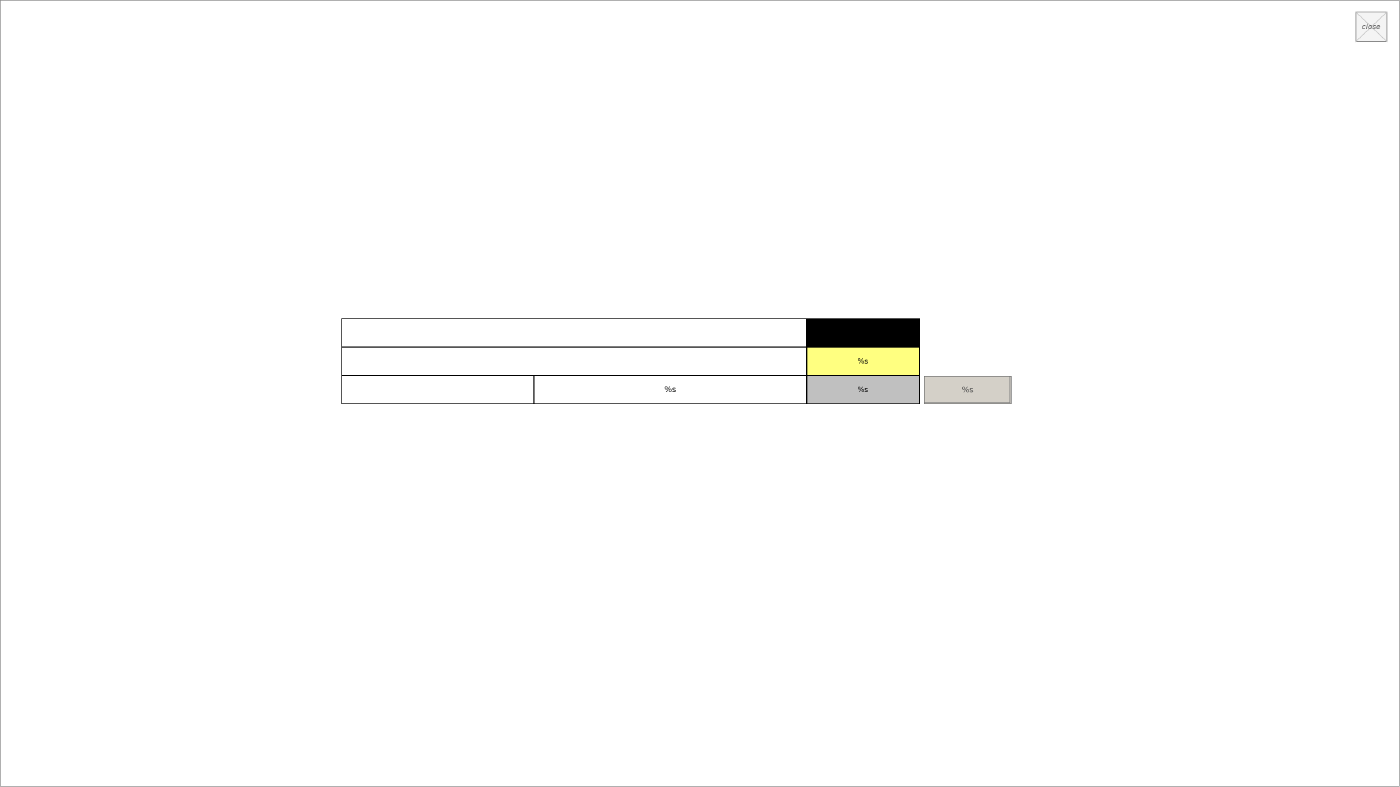
VISUALIZATION VISU_CONFIG_ECOMODE  // 1920x1080, background image fond_blanc_1280_1024
    Rectangle (468,476 638x39), text list: 'TextList_EcoMode', text index: 1
    Rectangle (468,437 638x39), text list: 'TextList_EcoMode', text index: 0
    Rectangle (468,515 264x39), text list: 'TextList_EcoMode', text index: 2
    Rectangle (1106,476 155x39), "%s", text variable: .MACHINE.CONF_Tps_Inactivite, input disabled if: NOT Global_Variables.PRG_USER.ACTU_USER.CONF_MACHINE
        OnMouseClick: write the text variable via InputWithLimits, min 0
    Rectangle (1106,437 155x39), colour toggle: MACHINE.CONF_Standby_Auto, input disabled if: NOT Global_Variables.PRG_USER.ACTU_USER.CONF_MACHINE
        toggle MACHINE.CONF_Standby_Auto
    Rectangle (732,515 374x39), "%s", text variable: .MACHINE.PRM_PROCESS_WEEKEND
    Rectangle (1106,515 155x39), "%s", colour toggle: MACHINE.PRM_RECORD_WEEKEND, text list: 'TextList_EcoMode', text index: 3
    Button (1267,516 120x38), "%s", input disabled if: NOT Global_Variables.PRG_USER.ACTU_USER.CONF_MACHINE, text list: 'TextList_EcoMode', text index: 4
        tap MAIN.bStartVerif
        OnMouseClick: execute { .MACHINE.PRM_LAUNCHER_WEEKEND:=TRUE; }
    Image (1859,16 43x41), image: close
        tap Global_Variables.RQ_PARAM_SYSTEM
        OnMouseClick: toggle RQ_PARAM_SYSTEM
        OnMouseClick: change screen: SYN_PROC
END_VISUALIZATION

(* stored: Version 1.1.0.1, ProductVersion 3.1.4024.11
   Visu VISU_CONFIG_ECOMODE: Id {607c3197-3e75-47ab-99ea-4f8f0a15afd9} *)
